# EPICS substitutions: vacuum/MAIN_TRUNK/db/l424_agilent4uhv.substitutions
# Agilent4UHV substitutions file

file db/agilent4uhv.db
{
     pattern {LOCA,			DEV,			PORT,		ADDR,	TIMEOUT}
     		{HL4,			VL424_1,		4uhv_1,		0,		0.2}
     		{HL4,			VL424_2,		4uhv_2,		0,		0.2}
}

file db/agilent4uhv_alias.db
{
     pattern {LOCA,			DEV,			SUB1,				SUB2,				SUB3,					SUB4,				PORT,		ADDR,	TIMEOUT}
     		 {HL4,			VL424_1,		IP01:L424_Acc601,		IP02:L424_Acc602,		IP03:L424_Acc603,			IP04:L424_Acc604,		4uhv_1,		0,		0.2}
		 {HL4,			VL424_2,		IP05:L424_Acc605,		IP06:L424_Wave601,	IP07:L424_Kly601,			IP08:Empty,			4uhv_2,		0,		0.2}
}
